(* IEC 61131-3 sources: tfc-hmi/packages/tfc_mcp_server/test/compiler/fixtures/beckhoff, 4 files *)

(* ---- pragmas.st ---- *)
{attribute 'qualified_only'}
VAR_GLOBAL
  GVL_Main : INT;
  GVL_Counter : DINT;
END_VAR

{attribute 'pack_mode' := '1'}
TYPE ST_Packed :
STRUCT
  field1 : BYTE;
  field2 : DWORD;
  field3 : BOOL;
END_STRUCT
END_TYPE

(* ---- method_property.st ---- *)
FUNCTION_BLOCK FB_Heater
VAR
  _temperature : REAL;
  _setpoint : REAL;
  _output : REAL;
  _enabled : BOOL;
END_VAR
  IF _enabled THEN
    _output := (_setpoint - _temperature) * 0.5;
  ELSE
    _output := 0.0;
  END_IF;
END_FUNCTION_BLOCK

METHOD PUBLIC Start : BOOL
VAR_INPUT
  initialSetpoint : REAL;
END_VAR
  _setpoint := initialSetpoint;
  _enabled := TRUE;
  Start := TRUE;
END_METHOD

METHOD PUBLIC Stop : BOOL
  _enabled := FALSE;
  _output := 0.0;
  Stop := TRUE;
END_METHOD

PROPERTY PUBLIC Temperature : REAL
// GET accessor
GET
VAR
END_VAR
  Temperature := _temperature;
END_GET
// SET accessor
SET
VAR
END_VAR
  _temperature := Temperature;
END_SET
END_PROPERTY

(* ---- oop_motor.st ---- *)
INTERFACE ITF_Drive
  METHOD Start : BOOL
  END_METHOD

  METHOD Stop : BOOL
  END_METHOD

  PROPERTY Speed : REAL
END_INTERFACE

FUNCTION_BLOCK FB_Motor EXTENDS FB_Base IMPLEMENTS ITF_Drive
VAR_INPUT
  bStart : BOOL;
  rSetSpeed : REAL;
END_VAR
VAR_OUTPUT
  bRunning : BOOL;
  rActSpeed : REAL;
END_VAR
VAR
  _state : INT;
  _rampRate : REAL := 10.0;
END_VAR
  IF bStart AND NOT bRunning THEN
    _state := 1;
    bRunning := TRUE;
  END_IF;

  IF bRunning THEN
    IF rActSpeed < rSetSpeed THEN
      rActSpeed := rActSpeed + _rampRate;
    ELSIF rActSpeed > rSetSpeed THEN
      rActSpeed := rActSpeed - _rampRate;
    END_IF;
  END_IF;
END_FUNCTION_BLOCK

// METHOD definitions would be in separate XML nodes in TcPOU
// but for raw .st testing, inline them here

(* ---- exst_extensions.st ---- *)
PROGRAM ExstTest
VAR
  latchOn : BOOL;
  latchOff : BOOL;
  triggerSet : BOOL;
  triggerReset : BOOL;
  ptrVal : POINTER TO INT;
  refVal : REFERENCE TO REAL;
  someInt : INT;
  someReal : REAL;
  i : INT;
END_VAR
  // S= (set/latch) operator
  latchOn S= triggerSet;

  // R= (reset) operator
  latchOff R= triggerReset;

  // POINTER operations
  ptrVal := ADR(someInt);
  someInt := ptrVal^;

  // REFERENCE operations
  refVal REF= someReal;

  // CONTINUE in loop
  FOR i := 0 TO 10 DO
    IF i = 5 THEN
      CONTINUE;
    END_IF;
    someInt := someInt + i;
  END_FOR;
END_PROGRAM
